# B&R Automation Studio project Lab1
Automation Studio 4.5.2.102

## Configuration Config1

### Task classes (Cpu.sw)
```
Cyclic#4:
  Program <- Program.prg
Binaries: udbdef, TCData, ashwd, User, asfw, arconfig, sysconf, Role, ashwac, iomap
Libraries: MotorCtrl
```

### Hardware
```
4PP065_0571_P74 : 4PP065.0571-P74 v1.1.2.0
  Connector IF5:
    ActivateDevice = 1
  ConfigurationID = LabBR
  Simulation = 1
```

## Logical view

### Library Logical/Libraries/MotorCtrl (ANSIC)

#### Constants.var - Exported constants
```iecst
VAR CONSTANT
	New_Variable : REAL := 0.0;
END_VAR
```

#### MotorCtrl.fun - Exported functions and function blocks
```iecst
{REDUND_ERROR} FUNCTION_BLOCK FB_Integrator (*TODO: Add your comment here*) (*$GROUP=User,$CAT=User,$GROUPICON=User.png,$CATICON=User.png*)
	VAR_INPUT
		in : {REDUND_UNREPLICABLE} REAL;
	END_VAR
	VAR_OUTPUT
		out : REAL;
	END_VAR
	VAR
		dt : REAL;
		prevstate : REAL;
	END_VAR
END_FUNCTION_BLOCK

{REDUND_ERROR} FUNCTION_BLOCK FB_Regulator (*TODO: Add your comment here*) (*$GROUP=User,$CAT=User,$GROUPICON=User.png,$CATICON=User.png*)
	VAR_INPUT
		e : {REDUND_UNREPLICABLE} REAL;
	END_VAR
	VAR_OUTPUT
		u : REAL;
	END_VAR
	VAR
		k_p : REAL;
		k_i : REAL;
		integrator : FB_Integrator;
		iyOld : REAL;
		max_abs_value : REAL;
		dt : REAL;
		prevstate : REAL;
		state_back1 : REAL;
		sum : REAL;
		b : REAL;
		a : REAL;
		u_max : REAL;
	END_VAR
END_FUNCTION_BLOCK

{REDUND_ERROR} FUNCTION_BLOCK FB_Motor (*TODO: Add your comment here*) (*$GROUP=User,$CAT=User,$GROUPICON=User.png,$CATICON=User.png*)
	VAR_INPUT
		u : {REDUND_UNREPLICABLE} REAL;
	END_VAR
	VAR_OUTPUT
		w : REAL;
	END_VAR
	VAR
		prevstate : REAL;
		integrator : FB_Integrator;
		phi : REAL;
		ke : REAL;
		Tm : REAL;
		dt : REAL;
		state : REAL;
	END_VAR
END_FUNCTION_BLOCK
```

#### FB_Motor.c
```c
#include <bur/plctypes.h>
#ifdef __cplusplus
	extern "C"
	{
#endif
	#include "MotorCtrl.h"
#ifdef __cplusplus
	};
#endif
/* TODO: Add your comment here */
void FB_Motor(struct FB_Motor* inst)
{

	inst->integrator.out = inst->w;
	inst->integrator.in = (inst->u/inst->ke - inst->w) * (inst->dt/inst->Tm);
	FB_Integrator(&inst->integrator);
	inst->integrator.in = inst->w = inst->integrator.out;
	inst->integrator.in *= inst->dt;
	inst->integrator.out = inst->phi;
	FB_Integrator(&inst->integrator);
	inst->phi = inst->integrator.out;
}
```

#### FB_Regulator.c
```c
#include <bur/plctypes.h>
#ifdef __cplusplus
	extern "C"
	{
#endif
	#include "MotorCtrl.h"
#ifdef __cplusplus
	};
#endif
/* TODO: Add your comment here */
void FB_Regulator(struct FB_Regulator* inst)
{
	inst->a = inst->e * inst->k_p;
	inst->b = inst->e * inst->k_i * inst->dt;
	if (inst->a > inst->max_abs_value){
		inst->a = inst->max_abs_value;
	}
	if (inst->a < -inst->max_abs_value){
		inst->a = -inst->max_abs_value;
	}
	inst->integrator.in = inst->b + inst->iyOld;
	FB_Integrator(&inst->integrator);
	inst->sum = inst->a + inst->integrator.out;
	inst->u = inst->sum;
	if (inst->u > inst->max_abs_value){
		inst->u = inst->max_abs_value;
	}
	if (inst->u < -inst->max_abs_value){
		inst->u = -inst->max_abs_value;
	}

	inst->iyOld = inst->u - inst->sum;
}
```

#### FB_Integrator.c
```c
#include <bur/plctypes.h>
#ifdef __cplusplus
	extern "C"
	{
#endif
	#include "MotorCtrl.h"
#ifdef __cplusplus
	};
#endif
/* TODO: Add your comment here */
void FB_Integrator(struct FB_Integrator* inst)
{
	/*TODO: Add your code here*/
	inst->out = inst->in * inst->dt + inst->prevstate;
	inst->prevstate = inst->out;
}
```

### Program Logical/Program

#### Variables.var
```iecst
VAR
	k : REAL;
	fb_motor1 : FB_Motor;
	fb_motor2 : FB_Motor;
	fb_regulator1 : FB_Regulator;
	fb_integrator1 : FB_Integrator;
	ke : REAL;
	Tm : REAL;
	Tj : REAL;
	speed : REAL;
	dt : REAL;
	enable : BOOL;
	flag : BOOL;
	counter : UDINT;
END_VAR
```

#### Cyclic.c
```c
#include <bur/plctypes.h>

#ifdef _DEFAULT_INCLUDES
	#include <AsDefault.h>
#endif

void _CYCLIC ProgramCyclic(void)
{
	if (enable){

		if (counter % 50 == 0)
		{
			flag = !flag;
			if (flag)
			{
				speed = 50;
			}
			else
			{
				speed = 0;
			}
		}
		fb_regulator1.e = speed - fb_motor1.w;
		FB_Regulator(&fb_regulator1);
		fb_motor1.u = fb_regulator1.u;
		FB_Motor(&fb_motor1);
		fb_motor2.u = speed * fb_motor2.ke;
		FB_Motor(&fb_motor2);
		counter += 1;

	}

}
```

#### Init.c
```c
#include <bur/plctypes.h>

#ifdef _DEFAULT_INCLUDES
	#include <AsDefault.h>
#endif

void _INIT ProgramInit(void)
{
	//Мотор Brush DC Motors 16C18 205.67
	dt = 0.1;
	Tj = 0.2*dt;
	Tm = 0.060;
	ke = 0.070;

	fb_regulator1.dt = dt;
	fb_regulator1.integrator.dt = dt;
	fb_regulator1.max_abs_value = 24.0;
	fb_regulator1.k_p = ke*Tm/Tj ;
	fb_regulator1.k_i = ke/Tj;
	fb_motor1.dt = dt;
	fb_motor1.integrator.dt = dt;
	fb_motor1.Tm = Tm;
	fb_motor1.ke = ke;
	fb_motor1.u = 0;
	fb_motor2.dt = dt;
	fb_motor2.integrator.dt = dt;
	fb_motor2.Tm = Tm;
	fb_motor2.ke = ke;
	fb_motor2.u = 0;
	counter = 0;
	speed = 0;
	enable = 1;
	flag = 0;
}
```

Listed in the project but not available here: Logical/Libraries/MotorCtrl/Types.typ
